(* CoDeSys 2.3.9.59 project: PD1.pro *)
(* Libraries: Standard.lib, SYSLIBCALLBACK.LIB *)

(* PLC configuration (modules and I/O channels)
Configuration EC4P-200 [Root] node -1, in %IB0 out %QB0 {EC4P_RestartPwrOn = WARMSTART; EC4P_MaxCycleTime = 20; EC4P_Com1BaudRate = 38400; EC4P_CAN1BaudRate = 125KBaud; EC4P_RoutingId = 127; EC4P_EasyNetId = 1; EC4P_EasyNetCfg = 0; EC4P_EasyNetCycleTime = 50; EC4P_RoutingChannel = CAN1; EC4P_IPFlags = 0; EC4P_IPAddress = 0; EC4P_SubNetMask = 0; EC4P_DefaultGateway = 0; EC4P_SummerWinterFlags = 0; EC4P_SummerWinterRule1 = 0; EC4P_SummerWinterRule2 = 0}
  Local I/O [EC4P_LocalIO] node 0, in %IB0 out %QB0 {EC4P_LocalInt = 0}
    I1 AT %IX0.0 [LocalBitInput] Input I1
    I2 AT %IX0.1 [LocalBitInput] Input I2
    I3 AT %IX0.2 [LocalBitInput] Input I3
    I4 AT %IX0.3 [LocalBitInput] Input I4
    I5 AT %IX0.4 [LocalBitInput] Input I5
    I6 AT %IX0.5 [LocalBitInput] Input I6
    I7 AT %IX0.6 [LocalBitInput] Input I7
    I8 AT %IX0.7 [LocalBitInput] Input I8
    I9 AT %IX1.0 [LocalBitInput] Input I9
    I10 AT %IX1.1 [LocalBitInput] Input I10
    I11 AT %IX1.2 [LocalBitInput] Input I11
    I12 AT %IX1.3 [LocalBitInput] Input I12
    I13 AT %IX1.4 [LocalDiagInput] Diagnostic Input I13
    I14 AT %IX1.5 [LocalDiagInput] Diagnostic Input I14
    I15 AT %IX1.6 [LocalDiagInput] Diagnostic Input I15
    I16 AT %IX1.7 [LocalDiagInput] Diagnostic Input I16
    I7_Analog AT %IW2 [LocalAnalogIn] Input I7, 10Bit, 0-10VDC
    I8_Analog AT %IW4 [LocalAnalogIn] Input I8, 10Bit, 0-10VDC
    I11_Analog AT %IW6 [LocalAnalogIn] Input I11, 10Bit, 0-10VDC
    I12_Analog AT %IW8 [LocalAnalogIn] Input I12, 10Bit, 0-10VDC
    Transistor Outputs [EC4P_TOutputs] node 0, in %IB10 out %QB0
      Q1 AT %QX0.0 [LocalBitOutput] Transistor-Output Q1
      Q2 AT %QX0.1 [LocalBitOutput] Transistor-Output Q2
      Q3 AT %QX0.2 [LocalBitOutput] Transistor-Output Q3
      Q4 AT %QX0.3 [LocalBitOutput] Transistor-Output Q4
      Q5 AT %QX0.4 [LocalBitOutput] Transistor-Output Q5
      Q6 AT %QX0.5 [LocalBitOutput] Transistor-Output Q6
      Q7 AT %QX0.6 [LocalBitOutput] Transistor-Output Q7
      Q8 AT %QX0.7 [LocalBitOutput] Transistor-Output Q8
    No Analog Output [EC4P_NoAnalogOutput] node 1, in %IB10 out %QB1
    No Keys [EC4P_NoKeys] node 2, in %IB10 out %QB1
    No Counter [EC4P_NoCounter] node 3, in %IB10 out %QB1
  Extension [EC4P_Extension] node 1, in %IB10 out %QB1
    No Extension [EC4P_NoExtension] node 0, in %IB10 out %QB1
*)

(* POU PLC_PRG, LD *)
PROGRAM PLC_PRG
VAR
END_VAR
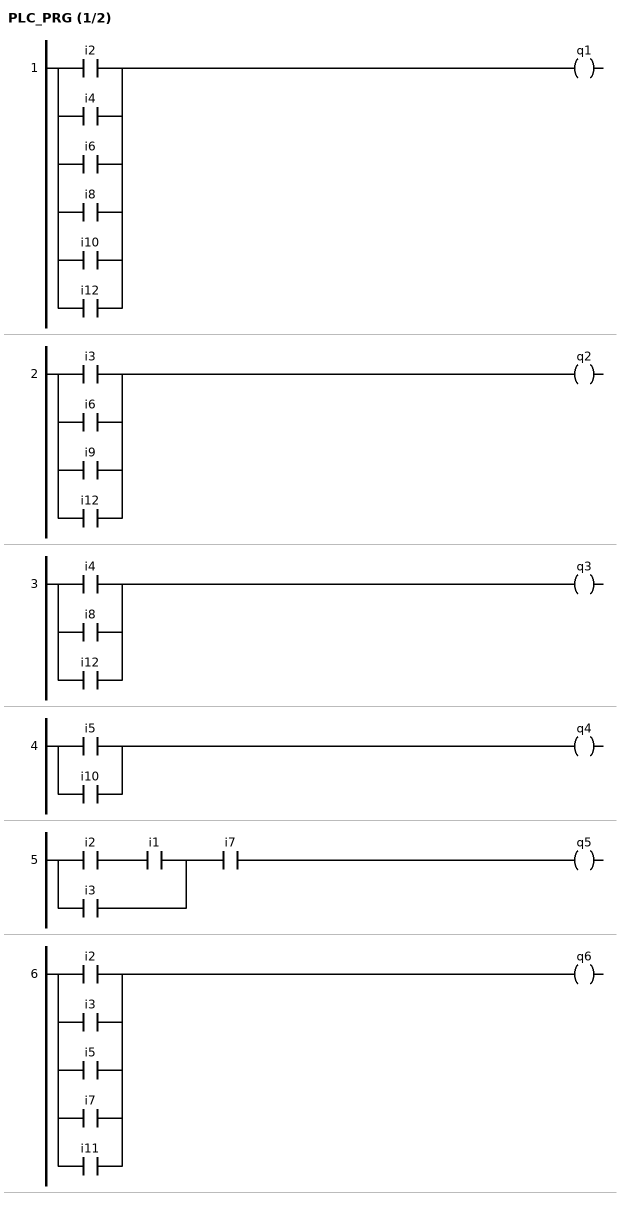
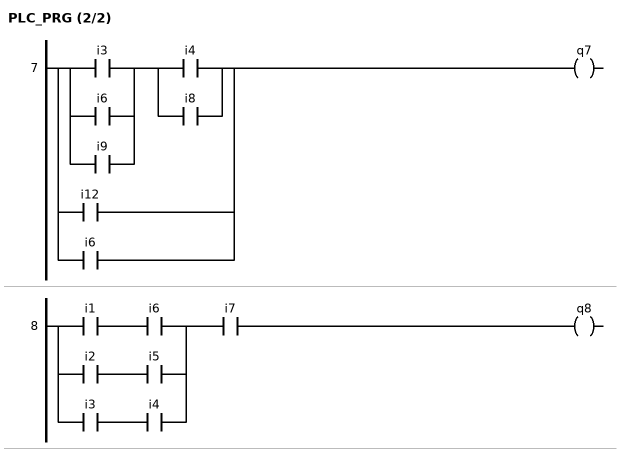
_LD_ (* Ladder Diagram *)
NETWORK 1
	{ [i2] | [i4] | [i6] | [i8] | [i10] | [i12] } --- (q1)
NETWORK 2
	{ [i3] | [i6] | [i9] | [i12] } --- (q2)
NETWORK 3
	{ [i4] | [i8] | [i12] } --- (q3)
NETWORK 4
	{ [i5] | [i10] } --- (q4)
NETWORK 5
	{ [i2] - [i1] | [i3] } - [i7] --- (q5)
NETWORK 6
	{ [i2] | [i3] | [i5] | [i7] | [i11] } --- (q6)
NETWORK 7
	{ { [i3] | [i6] | [i9] } - { [i4] | [i8] } | [i12] | [i6] } --- (q7)
NETWORK 8
	{ [i1] - [i6] | [i2] - [i5] | [i3] - [i4] } - [i7] --- (q8)
_END_LD_
(* the same logic as Structured Text *)
(* Network 1 *)
q1 := i2 OR i4 OR i6 OR i8 OR i10 OR i12;
(* Network 2 *)
q2 := i3 OR i6 OR i9 OR i12;
(* Network 3 *)
q3 := i4 OR i8 OR i12;
(* Network 4 *)
q4 := i5 OR i10;
(* Network 5 *)
q5 := (i2 AND i1 OR i3) AND i7;
(* Network 6 *)
q6 := i2 OR i3 OR i5 OR i7 OR i11;
(* Network 7 *)
q7 := (i3 OR i6 OR i9) AND (i4 OR i8) OR i12 OR i6;
(* Network 8 *)
q8 := (i1 AND i6 OR i2 AND i5 OR i3 AND i4) AND i7;
END_PROGRAM
